{attribute 'qualified_only'}
VAR_GLOBAL
IX_START AT %I*: BOOL;
IX_STOP AT %I*:	BOOL;
IW_VGR_CounterValueVertical  		AT %I* : UINT;
IW_VGR_CounterValueHorizontal  		AT %I* : UINT;
IW_VGR_CounterValueRotate  			AT %I* : UINT;

END_VAR

(* stored: Version 1.1.0.1, ProductVersion 3.1.4024.12
   GVL INPUT: Id {317528c4-17d9-4d6e-84cc-04007afaa00c} *)
